PROGRAM PRG_TEST
VAR
	fb_Max_Value_Test : FB_Max_Value_Test;
END_VAR

TcUnit.RUN();

END_PROGRAM

(* stored: Version 1.1.0.1, ProductVersion 3.1.4024.13
   POU PRG_TEST: Id {6e915b6b-d635-4ca5-ad05-73f49eb5e09a}, SpecialFunc None *)
